// TIA Portal V17 export
// export: Created 2025-08-05T09:35:56.5049697Z, ExportSetting WithDefaults, DisplayName Totally Integrated Automation Portal, DisplayVersion V17, DisplayName TIA Portal Openness, DisplayVersion V17, DisplayName TIA Portal Version Control Interface, DisplayVersion V17, DisplayName SINAMICS Startdrive Advanced, DisplayVersion V17, DisplayName SINAMICS Startdrive G130, G150, S120, S150, SINAMICS MV, S210, DisplayVersion V17, DisplayName SINAMICS Startdrive G110M, G120, G120C, G120D, G120P, G115D, DisplayVersion V17, DisplayName STEP 7 Professional, DisplayVersion V17, DisplayName STEP 7 Safety, DisplayVersion V17, DisplayName WinCC Advanced, DisplayVersion V17
FUNCTION_BLOCK "Control"   // FB266, LAD
{ S7_Optimized_Access := 'FALSE' }
VERSION : 0.1
// stored: AutoNumber true, IsIECCheckEnabled false, SetENOAutomatically false, UDAEnableTagReadback false
   VAR_INPUT
      iGraph_Step_1 : Bool;
      iInstance_Index : DInt;
   END_VAR
   VAR_IN_OUT
      ioGraph_Job_Select : Int;
   END_VAR
   VAR DB_SPECIFIC
      sStep : DInt;
      sNo_Faults_Active : Bool;
      Step_Delay { S7_SetPoint := 'True'} : TON_TIME;
      sCounter_Done : Bool;
      sCTU : IEC_COUNTER;
      sWeldJob { S7_SetPoint := 'True'} : Byte;
      sDelayDone : Bool;
   END_VAR
   VAR_TEMP   // added for the SCL form of the ladder/FBD networks
      _w1 : Bool;
      _w2 : Bool;
   END_VAR
BEGIN

REGION Network 1: Tooling Delay
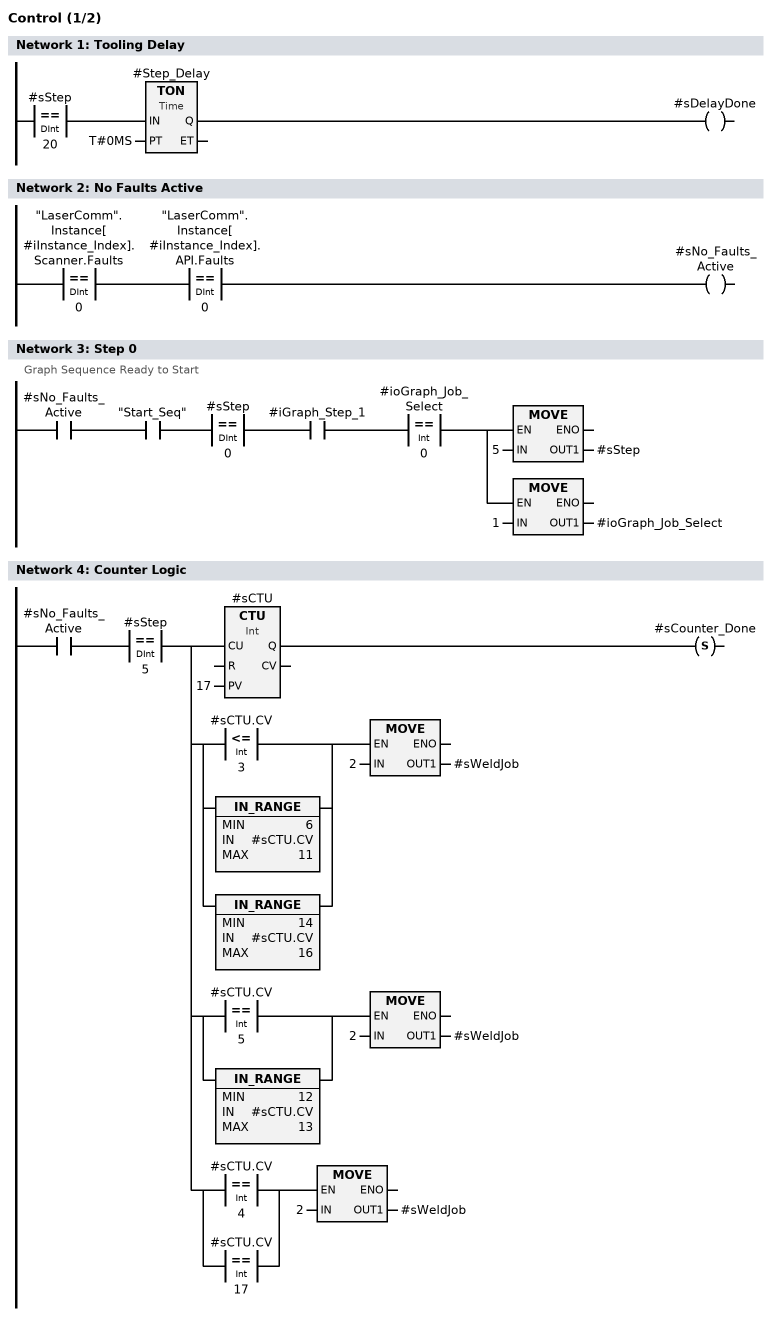
   RUNG wire#powerrail
      { S7_Templates := "SrcType := DInt" } EQ_Contact(in1 := #sStep, in2 := 20)
      { S7_Templates := "time_type := Time" } #Step_Delay.TON(pt := T#0MS, et =>)
      Coil( #sDelayDone )
   END_RUNG
   // the same network as SCL:
   #Step_Delay(IN := #sStep = 20, PT := T#0MS);   // TON
   #sDelayDone := #Step_Delay.Q;
END_REGION

REGION Network 2: No Faults Active
   RUNG wire#powerrail
      { S7_Templates := "SrcType := DInt" } EQ_Contact(in1 := "LaserComm".Instance[#iInstance_Index].Scanner.Faults, in2 := 0)
      { S7_Templates := "SrcType := DInt" } EQ_Contact(in1 := "LaserComm".Instance[#iInstance_Index].API.Faults, in2 := 0)
      Coil( #sNo_Faults_Active )
   END_RUNG
   // the same network as SCL:
   #sNo_Faults_Active := ("LaserComm".Instance[#iInstance_Index].Scanner.Faults = 0) AND ("LaserComm".Instance[#iInstance_Index].API.Faults = 0);
END_REGION

REGION Network 3: Step 0
   // Graph Sequence Ready to Start
   RUNG wire#powerrail
      Contact( #sNo_Faults_Active )
      Contact( "Start_Seq" )
      { S7_Templates := "SrcType := DInt" } EQ_Contact(in1 := #sStep, in2 := 0)
      Contact( #iGraph_Step_1 )
      { S7_Templates := "SrcType := Int" } EQ_Contact(in1 := #ioGraph_Job_Select, in2 := 0)
      wire#w1
      { S7_GenerateENO := "TRUE" } Move(in := 5, out1 => #sStep)
   END_RUNG
   RUNG wire#w1
      { S7_GenerateENO := "TRUE" } Move(in := 1, out1 => #ioGraph_Job_Select)
   END_RUNG
   // the same network as SCL:
   #_w1 := #sNo_Faults_Active AND "Start_Seq" AND (#sStep = 0) AND #iGraph_Step_1 AND (#ioGraph_Job_Select = 0);
   IF #_w1 THEN
       #sStep := 5;
       #ioGraph_Job_Select := 1;
   END_IF;
END_REGION

REGION Network 4: Counter Logic
   RUNG wire#powerrail
      Contact( #sNo_Faults_Active )
      { S7_Templates := "SrcType := DInt" } EQ_Contact(in1 := #sStep, in2 := 5)
      wire#w1
      { S7_Templates := "value_type := Int" } #sCTU.CTU(r :=, pv := 17, cv =>)
      S_Coil( #sCounter_Done )
   END_RUNG
   RUNG wire#w1
      { S7_Templates := "SrcType := Int" } LE_Contact(in1 := #sCTU.CV, in2 := 3)
      wire#w2
      Move(in := 2, out1 => #sWeldJob)
   END_RUNG
   RUNG wire#w1
      { S7_Templates := "SrcType := Int" } InRange(min := 6, in := #sCTU.CV, max := 11)
   END_RUNG wire#w2
   RUNG wire#w1
      { S7_Templates := "SrcType := Int" } InRange(min := 14, in := #sCTU.CV, max := 16)
   END_RUNG wire#w2
   RUNG wire#w1
      { S7_Templates := "SrcType := Int" } EQ_Contact(in1 := #sCTU.CV, in2 := 5)
      wire#w3
      Move(in := 2, out1 => #sWeldJob)
   END_RUNG
   RUNG wire#w1
      { S7_Templates := "SrcType := Int" } InRange(min := 12, in := #sCTU.CV, max := 13)
   END_RUNG wire#w3
   RUNG wire#w1
      { S7_Templates := "SrcType := Int" } EQ_Contact(in1 := #sCTU.CV, in2 := 4)
      wire#w4
      Move(in := 2, out1 => #sWeldJob)
   END_RUNG
   RUNG wire#w1
      { S7_Templates := "SrcType := Int" } EQ_Contact(in1 := #sCTU.CV, in2 := 17)
   END_RUNG wire#w4
   // the same network as SCL:
   #_w1 := #sNo_Faults_Active AND (#sStep = 5);
   #sCTU.CTU(CU := #_w1, PV := 17);
   IF #sCTU.Q THEN #sCounter_Done := TRUE; END_IF;
   IF #_w1 AND ((#sCTU.CV <= 3) OR ((6 <= #sCTU.CV) AND (#sCTU.CV <= 11)) OR ((14 <= #sCTU.CV) AND (#sCTU.CV <= 16))) THEN
       #sWeldJob := 2;
   END_IF;
   IF #_w1 AND ((#sCTU.CV = 5) OR ((12 <= #sCTU.CV) AND (#sCTU.CV <= 13))) THEN #sWeldJob := 2; END_IF;
   IF #_w1 AND ((#sCTU.CV = 4) OR (#sCTU.CV = 17)) THEN #sWeldJob := 2; END_IF;
END_REGION

REGION Network 5: Step 5
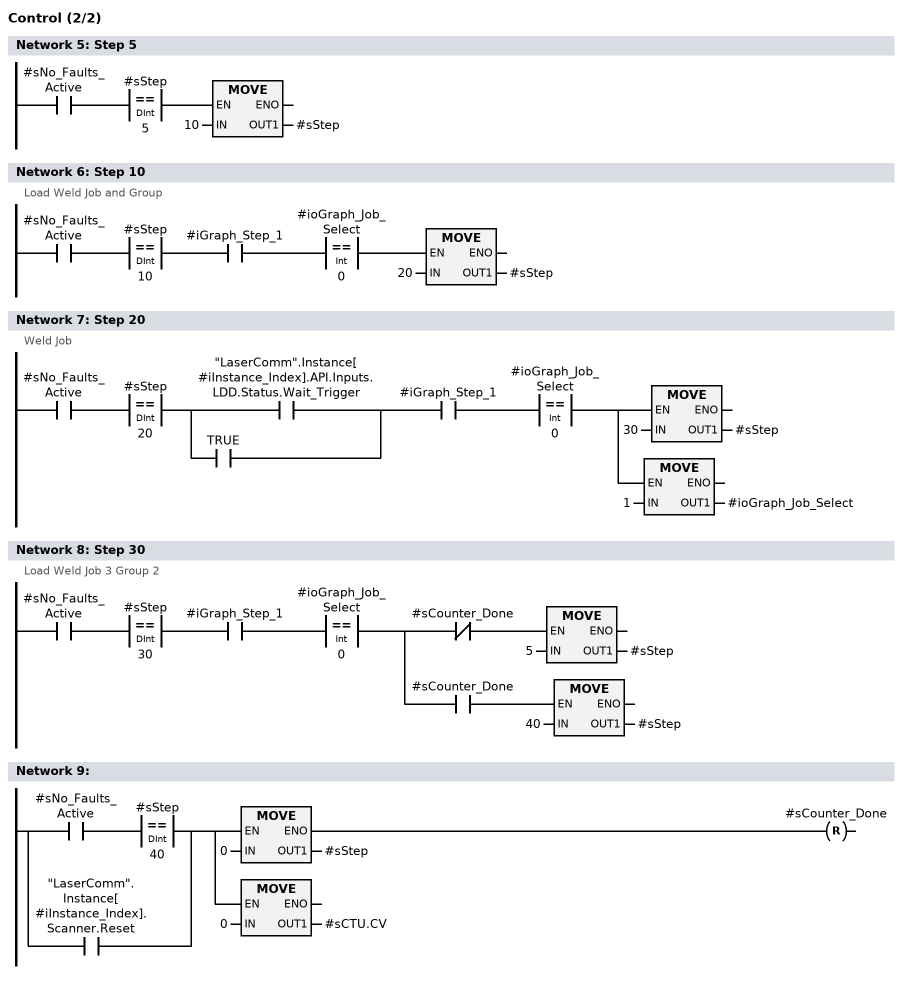
   RUNG wire#powerrail
      Contact( #sNo_Faults_Active )
      { S7_Templates := "SrcType := DInt" } EQ_Contact(in1 := #sStep, in2 := 5)
      { S7_GenerateENO := "TRUE" } Move(in := 10, out1 => #sStep)
   END_RUNG
   // the same network as SCL:
   IF #sNo_Faults_Active AND (#sStep = 5) THEN #sStep := 10; END_IF;
END_REGION

REGION Network 6: Step 10
   // Load Weld Job and Group
   RUNG wire#powerrail
      Contact( #sNo_Faults_Active )
      { S7_Templates := "SrcType := DInt" } EQ_Contact(in1 := #sStep, in2 := 10)
      Contact( #iGraph_Step_1 )
      { S7_Templates := "SrcType := Int" } EQ_Contact(in1 := #ioGraph_Job_Select, in2 := 0)
      { S7_GenerateENO := "TRUE" } Move(in := 20, out1 => #sStep)
   END_RUNG
   // the same network as SCL:
   IF #sNo_Faults_Active AND (#sStep = 10) AND #iGraph_Step_1 AND (#ioGraph_Job_Select = 0) THEN
       #sStep := 20;
   END_IF;
END_REGION

REGION Network 7: Step 20
   // Weld Job
   RUNG wire#powerrail
      Contact( #sNo_Faults_Active )
      { S7_Templates := "SrcType := DInt" } EQ_Contact(in1 := #sStep, in2 := 20)
      wire#w1
      Contact( "LaserComm".Instance[#iInstance_Index].API.Inputs.LDD.Status.Wait_Trigger )
      wire#w2
      Contact( #iGraph_Step_1 )
      { S7_Templates := "SrcType := Int" } EQ_Contact(in1 := #ioGraph_Job_Select, in2 := 0)
      wire#w3
      { S7_GenerateENO := "TRUE" } Move(in := 30, out1 => #sStep)
   END_RUNG
   RUNG wire#w1
      Contact( TRUE )
   END_RUNG wire#w2
   RUNG wire#w3
      { S7_GenerateENO := "TRUE" } Move(in := 1, out1 => #ioGraph_Job_Select)
   END_RUNG
   // the same network as SCL:
   #_w1 := #sNo_Faults_Active AND (#sStep = 20) AND ("LaserComm".Instance[#iInstance_Index].API.Inputs.LDD.Status.Wait_Trigger OR TRUE) AND #iGraph_Step_1 AND (#ioGraph_Job_Select = 0);
   IF #_w1 THEN
       #sStep := 30;
       #ioGraph_Job_Select := 1;
   END_IF;
END_REGION

REGION Network 8: Step 30
   // Load Weld Job 3 Group 2
   RUNG wire#powerrail
      Contact( #sNo_Faults_Active )
      { S7_Templates := "SrcType := DInt" } EQ_Contact(in1 := #sStep, in2 := 30)
      Contact( #iGraph_Step_1 )
      { S7_Templates := "SrcType := Int" } EQ_Contact(in1 := #ioGraph_Job_Select, in2 := 0)
      wire#w1
      I_Contact( #sCounter_Done )
      { S7_GenerateENO := "TRUE" } Move(in := 5, out1 => #sStep)
   END_RUNG
   RUNG wire#w1
      Contact( #sCounter_Done )
      { S7_GenerateENO := "TRUE" } Move(in := 40, out1 => #sStep)
   END_RUNG
   // the same network as SCL:
   #_w1 := #sNo_Faults_Active AND (#sStep = 30) AND #iGraph_Step_1 AND (#ioGraph_Job_Select = 0);
   IF #_w1 AND NOT #sCounter_Done THEN #sStep := 5; END_IF;
   IF #_w1 AND #sCounter_Done THEN #sStep := 40; END_IF;
END_REGION

REGION Network 9
   RUNG wire#powerrail
      Contact( #sNo_Faults_Active )
      { S7_Templates := "SrcType := DInt" } EQ_Contact(in1 := #sStep, in2 := 40)
      wire#w1
      { S7_GenerateENO := "TRUE" } Move(in := 0, out1 => #sStep)
      R_Coil( #sCounter_Done )
   END_RUNG
   RUNG wire#powerrail
      Contact( "LaserComm".Instance[#iInstance_Index].Scanner.Reset )
   END_RUNG wire#w1
   RUNG wire#w1
      { S7_GenerateENO := "TRUE" } Move(in := 0, out1 => #sCTU.CV)
   END_RUNG
   // the same network as SCL:
   // ENO of a box is taken as its EN; it also drops when the box reports an error
   #_w1 := (#sNo_Faults_Active AND (#sStep = 40)) OR "LaserComm".Instance[#iInstance_Index].Scanner.Reset;
   #_w2 := (#sNo_Faults_Active AND (#sStep = 40)) OR "LaserComm".Instance[#iInstance_Index].Scanner.Reset;
   IF #_w2 THEN
       #sStep := 0;
       #sCounter_Done := FALSE;
   END_IF;
   IF #_w1 THEN #sCTU.CV := 0; END_IF;
END_REGION
END_FUNCTION_BLOCK
